FUNCTION_BLOCK FB_AWEA
VAR_INPUT
END_VAR
VAR_OUTPUT
END_VAR
VAR
	DigIn		AT %I*		:ST_AWEA_In;
	DigOut		AT %Q*		:ST_AWEA_Out;
END_VAR

END_FUNCTION_BLOCK

(* stored: Version 1.1.0.1, ProductVersion 3.1.4024.11
   POU FB_AWEA: Id {4abb8e03-7980-4855-bec2-cd7833f94046}, SpecialFunc None *)
